(* IEC 61131-3 sources: s22-soft-shell/demos/rust_lib_usage/st_rust_demo1/st_testfiles, 2 files *)

(* ---- Calc_Test.st ---- *)
PROGRAM Calc_Test
    VAR
		a : Int;
		b : Int;
		c : bool;
		d : bool;
    END_VAR
		a := 3;
		b := 6;
		c := 3 >= a = 6-20 < 26; // Result = True
		d := ((16/4) = (b-4) * 2) xor c; // Result = False
END_PROGRAM

(* ---- Times2.st ---- *)
PROGRAM 07_Test_A
    VAR
		a : Int;
		b : Int;
		c : Int;
    END_VAR
		a := 2;
		b := a * 2;
		c := b * 2;
END_PROGRAM
